(* PLC project M3_24, Desconocido M3_22 1 *)
(* stored: creationDateTime 2025-05-15T11:40:54, modificationDateTime 2025-06-17T15:06:57 *)

PROGRAM Main
  VAR
    ArrayDatos : ARRAY[0..3] OF INT;
    iSuma : INT;
    ArrayPrueba : ARRAY[0..7] OF BOOL;
  END_VAR

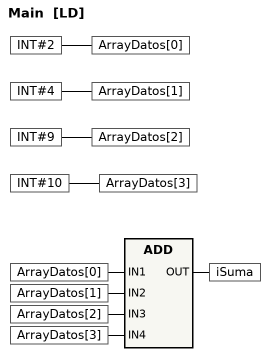
(* LD diagram, written out as Structured Text *)
ArrayDatos[0] := INT#2;
ArrayDatos[1] := INT#4;
ArrayDatos[2] := INT#9;
ArrayDatos[3] := INT#10;
iSuma := ArrayDatos[0] + ArrayDatos[1] + ArrayDatos[2] + ArrayDatos[3];
END_PROGRAM

CONFIGURATION Config0
  RESOURCE Res0 ON PLC
    TASK task0(INTERVAL := T#20ms, PRIORITY := 0);
    PROGRAM instance0 WITH task0 : Main;
  END_RESOURCE
END_CONFIGURATION
